{attribute 'qualified_only'}
{attribute 'pack_size' := '1'}
VAR_GLOBAL
	{region '__Chamber_Recipe_Body__' }
	RcipCMB			: ARRAY[0..100] OF scRCIP;		// Index 0 for Dummy
	{endregion}
 
	{region '__Chamber_Recipe_Profile__' }
	RcipARM			: ARRAY[0..100] OF WORD;		// Index 0 for Dummy
	{endregion}

END_VAR

(* stored: Version 1.1.0.1, ProductVersion 3.1.4024.16
   GVL gRCIP: Id {4dd80979-f07f-4854-a16c-7aead9c158e3} *)
